Staubli VAL3: tool.pjx

--- tool.pjx ---
Parameters version=s7.5 stackSize=5000 millimeterUnit=true
Program file=checkPoint.pgx
Program file=compose.pgx
Program file=delete.pgx
Program file=findItem.pgx
Program file=getInstr.pgx
Program file=getName.pgx
Program file=getSize.pgx
Program file=getTool.pgx
Program file=goToPoint.pgx
Program file=here.pgx
Program file=new.pgx
Program file=save.pgx
Program file=setInstr.pgx
Program file=setName.pgx
Program file=setTool.pgx
Data file=tool.dtx
Library alias=saveData path=Disk://saveData/saveData.pjx
Library alias=use path=Disk://kernel/userPage/userPage.pjx
Library alias=language path=Disk://kernel/language/language.pjx
Type name=InstrItem path=Disk://kernel/template/InstrItem/InstrItem.pjx
Type name=ToolItem path=Disk://kernel/template/ToolItem/ToolItem.pjx
Type name=TrajectoryItem path=Disk://kernel/template/TrajectoryItem/TrajectoryItem.pjx

--- checkPoint.pgx ---
public program checkPoint(bool& x_bCheck[])
begin
  x_bCheck=saveData:bCheck
end

--- compose.pgx ---
public program compose(num x_nIndexTool)
  local trsf tPar
  local tool tGun
  local point pPoint
begin
  pPoint=here(flange,world)
  tPar=!pPoint.trsf*saveData:rif2.trsf
  tGun.trsf=tPar
  call setTool(tGun,x_nIndexTool)
end

--- delete.pgx ---
public program delete(num x_nIndexTool)
begin
  delete(saveData:tData[x_nIndexTool])
end

--- findItem.pgx ---
public program findItem(InstrItem x_iItem, num& x_nResult)
  local num i
  local num l_nSize
  local num j
  local string l_sItem
  local string l_sMessage
  local num l_nResult
  local bool l_bFound
  local InstrItem l_iInstr[3]
  local string l_sSession
begin
  call getSize(l_nSize)
  // scan all the TCP for TCP ON OFF
  for i=0 to l_nSize-1
    call getName(l_sItem,i)
    //
    // SHOW THE TCP name
    //
    call saveData:getSession(l_sSession)
    l_sMessage="TCP "+l_sItem
    call use:typeLen(1,5,l_sMessage,38)
    call getInstr(l_iInstr,true,i)
    // scan deeper for all the action
    for j=0 to size(l_iInstr)-1
      // look inside
      l_bFound=(l_iInstr[j].sType==x_iItem.sType and(l_iInstr[j].sData==x_iItem.sData or find(l_iInstr[j].sData,x_iItem.sData+">")!=-1))
      // use nested items
      l_bFound=l_bFound or find(l_iInstr[j].sType+" "+l_iInstr[j].sData,x_iItem.sData+">")!=-1
      // FOUND IT
      if l_bFound
        x_nResult=-1
        call language:message(l_sMessage,23)
        popUpMsg(l_sMessage+x_iItem.sType+" "+x_iItem.sData+chr(10)+"TCP ON > "+l_iInstr[j].sType+" "+l_iInstr[j].sData)
        // back
        return
      endIf
    endFor
    call getInstr(l_iInstr,false,i)
    // scan deeper for all the action
    for j=0 to size(l_iInstr)-1
      // look inside
      l_bFound=(l_iInstr[j].sType==x_iItem.sType and find(l_iInstr[j].sData,x_iItem.sData)!=-1)
      // FOUND IT
      if l_bFound
        x_nResult=-1
        call language:message(l_sMessage,23)
        popUpMsg(l_sMessage+x_iItem.sType+" "+x_iItem.sData+chr(10)+"TCP OFF > "+l_sItem+" > "+l_iInstr[j].sType+" "+l_iInstr[j].sData)
        // back
        return
      endIf
    endFor
  endFor
end

--- getInstr.pgx ---
public program getInstr(InstrItem& x_iInstr[], bool x_bType, num x_nIndex)
  local string l_sInstruction
  local num i
begin
  // get the instruction and fill as an array
  if x_nIndex>=0
    if x_bType
      // take gun ON
      //resize(x_iInstr,1,size(saveData:tData[x_nIndex].iActionON))
      for i=0 to size(x_iInstr)-1
        x_iInstr[i]=saveData:tData[x_nIndex].iActionON[i]
      endFor
    else
      // take gun OFF
      //resize(x_iInstr,1,size(saveData:tData[x_nIndex].iActionOFF))
      for i=0 to size(x_iInstr)-1
        x_iInstr[i]=saveData:tData[x_nIndex].iActionOFF[i]
      endFor
    endIf
  endIf
end

--- getName.pgx ---
public program getName(string& x_sName[], num x_nIndex)
begin
  x_sName=saveData:tData[x_nIndex].name
end

--- getSize.pgx ---
public program getSize(num& nSize[])
begin
  nSize=size(saveData:tData)
end

--- getTool.pgx ---
public program getTool(tool& x_tTool[], num x_nIndex)
begin
  // get the tool
  x_tTool=saveData:tData[x_nIndex].tcp
end

--- goToPoint.pgx ---
public program goToPoint(num x_nIndexTool)
begin
  resetMotion()
  if x_nIndexTool==0
    movej(saveData:rif2,saveData:tData[x_nIndexTool].tcp,{25,25,25,9999,9999,off,50,50})
  else
    pPoint.trsf=position(saveData:rif2,world)
    pPoint.config={sfree,efree,wfree}
    movej(pPoint,saveData:tData[x_nIndexTool].tcp,{25,25,25,9999,9999,off,50,50})
  endIf
end

--- here.pgx ---
public program here()
begin
  saveData:rif2=here(saveData:tData[0].tcp,world)
  saveData:bCheck=true
end

--- new.pgx ---
public program new(trsf& x_tTool[])
  local num l_nSize
  local tool l_tTool
begin
  // only fifo politic
  call getSize(l_nSize)
  // TRSF
  insert(saveData:tData[l_nSize])
  l_tTool.trsf=x_tTool
  call setTool(l_tTool,l_nSize)
end

--- save.pgx ---
public program save(num& x_nResult[])
  local num i
begin
  x_nResult=saveData:libSave()
end

--- setInstr.pgx ---
public program setInstr(InstrItem& x_iInstr[], num x_nIndex, bool x_bType)
  local string l_sInstruction
  local num i
begin
  // get the instruction and fill as an array
  if x_nIndex>=0
    // save the data
    if x_bType
      // take gun ON
      //resize(saveData:tData[x_nIndex].iActionON,1,size(x_iInstr))
      for i=0 to size(x_iInstr)-1
        saveData:tData[x_nIndex].iActionON[i]=x_iInstr[i]
      endFor
    else
      // take gun OFF
      //resize(saveData:tData[x_nIndex].iActionOFF,1,size(x_iInstr))
      for i=0 to size(x_iInstr)-1
        saveData:tData[x_nIndex].iActionOFF[i]=x_iInstr[i]
      endFor
    endIf
  endIf
end

--- setName.pgx ---
public program setName(string x_sName, num x_nIndex)
begin
  // set the name
  saveData:tData[x_nIndex].name=x_sName
end

--- setTool.pgx ---
public program setTool(tool x_tTool, num x_nIndex)
begin
  // define the tool
  saveData:tData[x_nIndex].tcp=flange
  saveData:tData[x_nIndex].tcp.trsf=x_tTool.trsf
  saveData:tData[x_nIndex].tcp.ctime=x_tTool.ctime
  saveData:tData[x_nIndex].tcp.otime=x_tTool.otime
end
